{attribute addProperty BoxType "EL3681-0000-0018"}
{attribute addProperty Id "Disable_autorangeBIT10.1251Start_calibrationBIT10.1252Mode_BIT_0BIT10.1255Mode_BIT_1BIT10.1255Mode_BIT_2BIT10.1255Mode_BIT_3BIT10.1255RangeSINT819"}
{attribute addProperty CRC "1268879839"}
{attribute addProperty SizeInBites "16"}
{attribute addProperty SizeInBytes "2"}
TYPE Control_4BA191DF :
STRUCT
	{attribute addProperty Name "Disable_autorange"}
	Disable_autorange : BIT;
	{attribute addProperty Name "Start_calibration"}
	Start_calibration : BIT;
	{attribute 'hide'}
	reserve_1_BIT_0 : BIT;
	{attribute 'hide'}
	reserve_1_BIT_1 : BIT;
	{attribute addProperty Name "Mode"}
	Mode_BIT_0 : BIT;
	{attribute addProperty Name "Mode"}
	Mode_BIT_1 : BIT;
	{attribute addProperty Name "Mode"}
	Mode_BIT_2 : BIT;
	{attribute addProperty Name "Mode"}
	Mode_BIT_3 : BIT;
	{attribute addProperty Name "Range"}
	Range : SINT;
END_STRUCT
END_TYPE

(* stored: Version 1.2.0.0, ProductVersion 3.1.4024.9
   DUT Control_4BA191DF: Id {d170966c-0e09-49bd-bd58-f3cb92a9312e} *)
